// TIA Portal V18 export
// export: Created 2026-06-22T11:43:40.7540758Z, ExportSetting WithDefaults, DisplayName Totally Integrated Automation Portal, DisplayVersion V18, DisplayName TIA Portal Openness, DisplayVersion V18, DisplayName TIA Portal Version Control Interface, DisplayVersion V18, DisplayName STEP 7 Professional, DisplayVersion V18, DisplayName STEP 7 Safety, DisplayVersion V18, DisplayName WinCC Professional, DisplayVersion V18
Screen "Screen_1"  1440x900, Number=2
  ScreenLayer 
    GraphicView "Graphic view_1" at 0,0 size 1440x900  Picture=Thiết kế chưa có tên (2)_1
    GraphicIOField "Graphic I/O field_9" at 430,521 size 275x288  Mode=InOutput, OnValue=1, PictureList=GL_BonChua_MucDich
    GraphicIOField "Graphic I/O field_10" at 154,90 size 233x295  Mode=InOutput, OnValue=1, PictureList=GL_BonTron_MucDich
    GraphicIOField "Graphic I/O field_2" at 904,517 size 275x288  Mode=InOutput, OnValue=1, PictureList=GL_BonChua_MucDich
    GraphicIOField "Graphic I/O field_3" at 486,90 size 233x295  Mode=InOutput, OnValue=1, PictureList=GL_BonTron_MucDich
    GraphicIOField "Graphic I/O field_4" at 811,89 size 233x295  Mode=InOutput, OnValue=1, PictureList=GL_BonTron_MucDich
    GraphicIOField "Graphic I/O field_6" at 1160,89 size 233x295  Mode=InOutput, OnValue=1, PictureList=GL_BonTron_MucDich
    GraphicView "Graphic view_3" at 201,61 size 11x113  Picture=Graphic_24
    GraphicIOField "Graphic I/O field_5" at 189,70 size 51x78  Mode=InOutput, OnValue=1, PictureList=GL_Van_NamDoc
    GraphicView "Graphic view_2" at 544,60 size 11x113  Picture=Graphic_24
    GraphicIOField "Graphic I/O field_12" at 533,70 size 51x78  Mode=InOutput, OnValue=1, PictureList=GL_Van_NamDoc
    GraphicView "Graphic view_4" at 869,59 size 11x113  Picture=Graphic_24
    GraphicIOField "Graphic I/O field_13" at 860,69 size 51x78  Mode=InOutput, OnValue=1, PictureList=GL_Van_NamDoc
    GraphicView "Graphic view_5" at 1204,58 size 11x117  Picture=Graphic_24
    GraphicIOField "Graphic I/O field_14" at 1193,67 size 51x78  Mode=InOutput, OnValue=1, PictureList=GL_Van_NamDoc
    GraphicView "Graphic view_6" at 229,330 size 11x172  Picture=Graphic_24
    GraphicIOField "Graphic I/O field_11" at 220,429 size 51x78  Mode=InOutput, OnValue=1, PictureList=GL_Van_NamDoc
    GraphicIOField "Graphic I/O field_8" at 220,339 size 51x78  Mode=InOutput, OnValue=1, PictureList=GL_Van_NamDoc
    GraphicView "Graphic view_7" at 568,331 size 11x211  Picture=Graphic_24
    GraphicView "Graphic view_8" at 869,328 size 11x164  Picture=Graphic_24
    GraphicView "Graphic view_9" at 1224,328 size 11x164  Picture=Graphic_24
    GraphicIOField "Graphic I/O field_15" at 556,341 size 51x78  Mode=InOutput, OnValue=1, PictureList=GL_Van_NamDoc
    GraphicIOField "Graphic I/O field_16" at 558,417 size 51x78  Mode=InOutput, OnValue=1, PictureList=GL_Van_NamDoc
    GraphicIOField "Graphic I/O field_18" at 857,346 size 51x78  Mode=InOutput, OnValue=1, PictureList=GL_Van_NamDoc
    GraphicIOField "Graphic I/O field_20" at 857,412 size 51x78  Mode=InOutput, OnValue=1, PictureList=GL_Van_NamDoc
    GraphicIOField "Graphic I/O field_19" at 1214,347 size 51x78  Mode=InOutput, OnValue=1, PictureList=GL_Van_NamDoc
    GraphicIOField "Graphic I/O field_21" at 1213,419 size 51x78  Mode=InOutput, OnValue=1, PictureList=GL_Van_NamDoc
    GraphicView "Graphic view_10" at 223,500 size 25x5  Picture=Graphic_25
    GraphicView "Graphic view_11" at 1216,490 size 25x5  Picture=Graphic_25
    GraphicView "Graphic view_12" at 223,523 size 25x5  Picture=Graphic_25
    GraphicView "Graphic view_13" at 1216,515 size 25x5  Picture=Graphic_25
    GraphicView "Graphic view_14" at 252,501 size 5x26  Picture=Graphic_24
    GraphicView "Graphic view_15" at 1206,492 size 5x26  Picture=Graphic_24
    GraphicView "Graphic view_16" at 254,510 size 242x11  Picture=Graphic_25
    GraphicView "Graphic view_17" at 487,513 size 11x57  Picture=Graphic_24
    GraphicView "Graphic view_18" at 521,159 size 11x19  Picture=Graphic_24
    GraphicView "Graphic view_19" at 440,157 size 90x11  Picture=Graphic_25
    GraphicView "Graphic view_20" at 437,160 size 11x408  Picture=Graphic_24
    GraphicView "Graphic view_21" at 231,560 size 213x11  Picture=Graphic_25
    GraphicView "Graphic view_22" at 228,525 size 11x44  Picture=Graphic_24
    GraphicView "Graphic view_23" at 630,485 size 248x11  Picture=Graphic_25
    GraphicView "Graphic view_24" at 626,488 size 11x75  Picture=Graphic_24
    GraphicView "Graphic view_25" at 640,503 size 11x68  Picture=Graphic_24
    GraphicView "Graphic view_26" at 644,501 size 566x11  Picture=Graphic_25
    GraphicView "Graphic view_27" at 1224,517 size 11x51  Picture=Graphic_24
    GraphicView "Graphic view_28" at 1142,560 size 90x11  Picture=Graphic_25
    GraphicView "Graphic view_29" at 1139,99 size 11x469  Picture=Graphic_24
    GraphicView "Graphic view_30" at 1005,93 size 143x11  Picture=Graphic_25
    GraphicView "Graphic view_31" at 1000,95 size 11x86  Picture=Graphic_24
    GraphicView "Graphic view_32" at 564,755 size 11x103  Picture=Graphic_24
    GraphicIOField "Graphic I/O field_24" at 554,759 size 51x78  Mode=InOutput, OnValue=1, PictureList=GL_Van_NamDoc
    GraphicView "Graphic view_33" at 567,849 size 22x11  Picture=Graphic_25
    GraphicView "Graphic view_34" at 581,833 size 11x40  Picture=Graphic_24
    GraphicView "Graphic view_36" at 132,426 size 8x44  Picture=Graphic_28
    GraphicView "Graphic view_35" at 133,425 size 103x6  Picture=Graphic_29
    GraphicIOField "Graphic I/O field_7" at 133,396 size 83x47  Mode=InOutput, OnValue=1, PictureList=GL_Van_NamNgang
    GraphicIOField "Graphic I/O field_33" at 282,542 size 60x42  Mode=InOutput, OnValue=1, PictureList=GL_Pump_ChuyenDich
    GraphicView "Graphic view_38" at 371,61 size 2x119  Picture=Graphic_24
    GraphicView "Graphic view_40" at 352,178 size 22x2  Picture=Graphic_25
    GraphicView "Graphic view_39" at 361,99 size 21x47  Picture=Graphic_32
    GraphicView "Graphic view_41" at 125,453 size 21x47  Picture=Graphic_32
    GraphicView "Graphic view_37" at 341,167 size 28x25  Picture=Graphic_34
    GraphicView "Graphic view_42" at 473,422 size 103x6  Picture=Graphic_29
    GraphicIOField "Graphic I/O field_17" at 471,394 size 83x47  Mode=InOutput, OnValue=1, PictureList=GL_Van_NamNgang
    GraphicView "Graphic view_43" at 472,423 size 8x44  Picture=Graphic_28
    GraphicView "Graphic view_44" at 466,451 size 21x47  Picture=Graphic_32
    GraphicView "Graphic view_45" at 872,415 size 108x6  Picture=Graphic_29
    GraphicIOField "Graphic I/O field_22" at 903,387 size 83x47  Mode=InOutput, OnValue=1, PictureList=GL_Van_NamNgang
    GraphicView "Graphic view_46" at 976,415 size 8x35  Picture=Graphic_28
    GraphicView "Graphic view_47" at 970,434 size 21x47  Picture=Graphic_32
    GraphicView "Graphic view_48" at 1226,422 size 118x6  Picture=Graphic_29
    GraphicIOField "Graphic I/O field_23" at 1257,394 size 83x47  Mode=InOutput, OnValue=1, PictureList=GL_Van_NamNgang
    GraphicView "Graphic view_49" at 1336,422 size 8x35  Picture=Graphic_28
    GraphicView "Graphic view_50" at 1331,441 size 21x47  Picture=Graphic_32
    GraphicView "Graphic view_51" at 709,59 size 2x119  Picture=Graphic_24
    GraphicView "Graphic view_52" at 1047,60 size 2x116  Picture=Graphic_24
    GraphicView "Graphic view_53" at 1387,60 size 2x114  Picture=Graphic_24
    GraphicView "Graphic view_54" at 700,102 size 21x47  Picture=Graphic_32
    GraphicView "Graphic view_55" at 1038,104 size 21x47  Picture=Graphic_32
    GraphicView "Graphic view_56" at 1378,106 size 21x47  Picture=Graphic_32
    GraphicView "Graphic view_57" at 689,177 size 22x2  Picture=Graphic_25
    GraphicView "Graphic view_58" at 1016,175 size 33x2  Picture=Graphic_25
    GraphicView "Graphic view_59" at 1366,173 size 22x2  Picture=Graphic_25
    GraphicView "Graphic view_60" at 672,166 size 28x25  Picture=Graphic_34
    GraphicView "Graphic view_61" at 1000,165 size 28x25  Picture=Graphic_34
    GraphicView "Graphic view_62" at 1347,162 size 28x25  Picture=Graphic_34
    GraphicView "Graphic view_63" at 584,865 size 16x11  Picture=Graphic_25
    GraphicView "Graphic view_64" at 584,830 size 159x11  Picture=Graphic_25
    GraphicView "Graphic view_65" at 598,858 size 5x26  Picture=Graphic_24
    GraphicView "Graphic view_66" at 603,858 size 5x26  Picture=Graphic_24
    GraphicView "Graphic view_67" at 605,866 size 68x11  Picture=Graphic_25
    GraphicIOField "Graphic I/O field_1" at 608,851 size 60x42  Mode=InOutput, OnValue=1, PictureList=GL_Pump_ChuyenDich
    GraphicView "Graphic view_68" at 668,858 size 5x26  Picture=Graphic_24
    GraphicView "Graphic view_69" at 674,858 size 5x26  Picture=Graphic_24
    GraphicView "Graphic view_70" at 675,866 size 13x11  Picture=Graphic_25
    GraphicView "Graphic view_71" at 682,513 size 11x361  Picture=Graphic_24
    GraphicIOField "Graphic I/O field_25" at 672,597 size 51x78  Mode=InOutput, OnValue=1, PictureList=GL_Van_NamDoc
    GraphicView "Graphic view_72" at 684,510 size 376x11  Picture=Graphic_25
    GraphicView "Graphic view_73" at 1053,512 size 11x26  Picture=Graphic_24
    GraphicIOField "Graphic I/O field_34" at 587,792 size 90x71  Mode=InOutput, OnValue=1, PictureList=GL_Pump_TuanHoanLoc
    GraphicView "Graphic view_74" at 735,752 size 11x144  Picture=Graphic_24
    GraphicIOField "Graphic I/O field_27" at 725,829 size 51x78  Mode=InOutput, OnValue=1, PictureList=GL_Van_NamDoc
    GraphicIOField "Graphic I/O field_26" at 725,757 size 51x78  Mode=InOutput, OnValue=1, PictureList=GL_Van_NamDoc
    GraphicView "Graphic view_75" at 739,889 size 528x11  Picture=Graphic_25
    GraphicView "Graphic view_76" at 738,748 size 65x11  Picture=Graphic_25
    GraphicView "Graphic view_77" at 799,521 size 11x236  Picture=Graphic_24
    GraphicView "Graphic view_78" at 801,518 size 211x11  Picture=Graphic_25
    GraphicView "Graphic view_79" at 1005,520 size 11x38  Picture=Graphic_24
    GraphicView "Graphic view_80" at 469,833 size 103x6  Picture=Graphic_29
    GraphicView "Graphic view_81" at 467,834 size 8x44  Picture=Graphic_28
    GraphicView "Graphic view_82" at 461,854 size 21x47  Picture=Graphic_32
    GraphicIOField "Graphic I/O field_30" at 467,804 size 83x47  Mode=InOutput, OnValue=1, PictureList=GL_Van_NamNgang
    GraphicView "Graphic view_83" at 1040,751 size 11x75  Picture=Graphic_24
    GraphicIOField "Graphic I/O field_28" at 1030,754 size 51x78  Mode=InOutput, OnValue=1, PictureList=GL_Van_NamDoc
    GraphicView "Graphic view_84" at 1042,818 size 62x11  Picture=Graphic_25
    GraphicView "Graphic view_85" at 1100,802 size 11x40  Picture=Graphic_24
    GraphicView "Graphic view_86" at 1104,800 size 103x11  Picture=Graphic_25
    GraphicIOField "Graphic I/O field_35" at 1108,764 size 90x71  Mode=InOutput, OnValue=1, PictureList=GL_Pump_TuanHoanLoc
    GraphicView "Graphic view_87" at 1103,833 size 12x11  Picture=Graphic_25
    GraphicView "Graphic view_88" at 1112,825 size 5x26  Picture=Graphic_24
    GraphicView "Graphic view_89" at 1117,825 size 5x26  Picture=Graphic_24
    GraphicView "Graphic view_90" at 1118,833 size 72x11  Picture=Graphic_25
    GraphicIOField "Graphic I/O field_36" at 1123,820 size 60x42  Mode=InOutput, OnValue=1, PictureList=GL_Pump_ChuyenDich
    GraphicView "Graphic view_91" at 1186,825 size 5x26  Picture=Graphic_24
    GraphicView "Graphic view_92" at 1192,825 size 5x26  Picture=Graphic_24
    GraphicView "Graphic view_93" at 1195,833 size 13x11  Picture=Graphic_25
    GraphicView "Graphic view_94" at 1201,589 size 11x252  Picture=Graphic_24
    GraphicIOField "Graphic I/O field_29" at 1191,655 size 51x78  Mode=InOutput, OnValue=1, PictureList=GL_Van_NamDoc
    GraphicIOField "Graphic I/O field_37" at 1156,541 size 60x42  Mode=InOutput, OnValue=1, PictureList=GL_Pump_ChuyenDich
    GraphicView "Graphic view_95" at 1204,587 size 150x11  Picture=Graphic_25
    GraphicView "Graphic view_96" at 1257,590 size 11x307  Picture=Graphic_24
    GraphicView "Graphic view_97" at 1345,589 size 11x192  Picture=Graphic_24
    GraphicView "Graphic view_98" at 1352,589 size 75x6  Picture=Graphic_29
    GraphicIOField "Graphic I/O field_32" at 1346,558 size 83x47  Mode=InOutput, OnValue=1, PictureList=GL_Van_NamNgang
    GraphicView "Graphic view_99" at 1420,591 size 8x35  Picture=Graphic_28
    GraphicView "Graphic view_100" at 1414,607 size 21x47  Picture=Graphic_32
    GraphicView "Graphic view_102" at 1368,50 size 41x72  Picture=Graphic_37
    GraphicView "Graphic view_103" at 1365,159 size 28x31  Picture=Graphic_38
    GraphicView "Graphic view_104" at 1027,50 size 41x72  Picture=Graphic_37
    GraphicView "Graphic view_105" at 690,50 size 41x72  Picture=Graphic_37
    GraphicView "Graphic view_106" at 352,50 size 41x72  Picture=Graphic_37
    GraphicView "Graphic view_107" at 352,121 size 41x74  Picture=Graphic_39
    GraphicView "Graphic view_108" at 691,121 size 41x74  Picture=Graphic_39
    GraphicView "Graphic view_109" at 1028,121 size 41x74  Picture=Graphic_39
    GraphicView "Graphic view_110" at 1368,119 size 41x74  Picture=Graphic_39
    GraphicView "Graphic view_101" at 1012,165 size 45x26  Picture=Graphic_40
    GraphicView "Graphic view_111" at 676,167 size 45x26  Picture=Graphic_40
    GraphicView "Graphic view_112" at 341,167 size 38x26  Picture=Graphic_40
    GraphicIOField "Graphic I/O field_38" at 123,84 size 292x298  Mode=Output, OnValue=1, PictureList=GL_Khuay_8Frame
    GraphicIOField "Graphic I/O field_39" at 459,83 size 292x298  Mode=InOutput, OnValue=1, PictureList=GL_Khuay_8Frame
    GraphicIOField "Graphic I/O field_40" at 782,86 size 292x298  Mode=InOutput, OnValue=1, PictureList=GL_Khuay_8Frame
    GraphicIOField "Graphic I/O field_41" at 1130,89 size 292x298  Mode=InOutput, OnValue=1, PictureList=GL_Khuay_8Frame
    GraphicView "Graphic view_113" at 1280,567 size 56x45  Picture=Graphic_44
    GraphicView "Graphic view_115" at 1338,606 size 28x43  Picture=Graphic_46
    GraphicView "Graphic view_114" at 1246,722 size 28x43  Picture=Graphic_46
    GraphicView "Graphic view_116" at 1340,714 size 33x47  Picture=Graphic_47
    GraphicView "Graphic view_117" at 1327,779 size 50x52  Picture=Graphic_48
    GraphicView "Graphic view_118" at 1341,815 size 21x47  Picture=Graphic_32
    GraphicView "Graphic view_119" at 1337,843 size 29x56  Picture=Graphic_49
    GraphicView "Graphic view_120" at 939,821 size 108x6  Picture=Graphic_29
    GraphicIOField "Graphic I/O field_31" at 930,792 size 83x47  Mode=InOutput, OnValue=1, PictureList=GL_Van_NamNgang
    GraphicView "Graphic view_121" at 934,821 size 8x44  Picture=Graphic_28
    GraphicView "Graphic view_122" at 929,842 size 21x47  Picture=Graphic_32
    IOField "I/O field_1" at 113,69 size 67x32  DataFormat=Decimal, FormatPattern=999999, Mode=InOutput
    GraphicView "Graphic view_123" at 775,636 size 55x48  Picture=Graphic_50
    IOField "I/O field_2" at 300,127 size 67x28  DataFormat=Decimal, FormatPattern=999999, Mode=InOutput
